% RSLogix 500 project GENERATO.RSS, saved by version 8.30.00.16 %
PROJECT "GENERATO"    % processor: Bul.1763 MicroLogix 1100 Series B %

PROGRAM FILES
  LAD 2   2 rungs

DATA FILES
  O0 OUTPUT  4 elements
  I1 INPUT  6 elements
  S2 STATUS  66 elements
  B3 BINARY  1 elements
  T4 TIMER  1 elements
  C5 COUNTER  1 elements
  R6 CONTROL  1 elements
  N7 INTEGER  1 elements
  F8 FLOAT  1 elements

LADDER 2
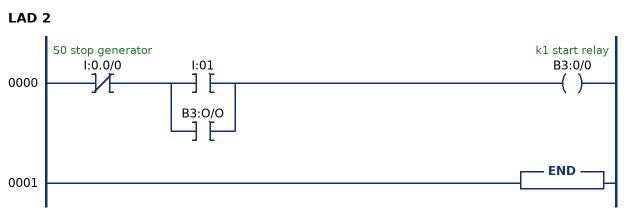
% Rung: 0 %  % edit flag set %
SOR XIO I:0.0/0 BST XIC I:01 NXB XIC B3:O/O BND OTE B3:0/0 EOR
%   I:0.0/0  "S0 stop generator" %
%   B3:0/0  "k1 start relay" %
% Rung: 1 %
SOR END EOR

OTHER DOCUMENTED ADDRESSES
  I:1  "S1 start generator"
